# EPICS substitutions: apps/mpodLvApp/Db/mmtb-lv.substitutions
file "db/mpod8008l.db" {
    pattern {HOST,CH,SCAN,PORT,DETALIAS}
{"%(mmtblv)","0","2 second","B_HW_MMTBLV_Sl0_Ch0","B_DET_SAMBA_LV_0"}
{"%(mmtblv)","1","2 second","B_HW_MMTBLV_Sl0_Ch1","B_DET_SAMBA_LV_1"}
{"%(mmtblv)","2","2 second","B_HW_MMTBLV_Sl0_Ch2","B_DET_SAMBA_LV_2"}
{"%(mmtblv)","3","2 second","B_HW_MMTBLV_Sl0_Ch3","B_DET_SAMBA_LV_3"}
{"%(mmtblv)","4","2 second","B_HW_MMTBLV_Sl0_Ch4","B_DET_SAMBA_LV_4"}
{"%(mmtblv)","5","2 second","B_HW_MMTBLV_Sl0_Ch5","B_DET_SAMBA_LV_5"}
}

file "db/mpod-crate.db" {
pattern { HOST }
        { mmtblv }
}
